// TwinCAT 3 PLC project Untitled1
// ProgramVersion: 3.1.4023.0
// libraries:
//   Tc2_Standard, * (Beckhoff Automation GmbH)
//   Tc2_System, * (Beckhoff Automation GmbH)
//   Tc2_Utilities, * (Beckhoff Automation GmbH)
//   Tc3_Module, * (Beckhoff Automation GmbH)
// project tree:
//   DUTs/ E_EventType.TcDUT, ST_Event.TcDUT
//   / PlcTask.TcTTO
//   POUs/ EventLogger.TcPOU, FB_CSVPersistentEventStorage.TcPOU, I_PersistentEventStorage.TcIO, MAIN.TcPOU, UpdateEventTimeStampWithSystemTime.TcPOU
// real-time tasks:
//   TASK PlcTask: cycle T#10ms, priority 20, ADS port 350

CONFIGURATION Untitled1
    RESOURCE PLC ON TwinCAT3
        TASK PlcTask(INTERVAL := T#10ms, PRIORITY := 20);
        PROGRAM MAIN WITH PlcTask : MAIN;
    END_RESOURCE
END_CONFIGURATION

// ---- DUTs/E_EventType.TcDUT
{attribute 'qualified_only'}
{attribute 'strict'}
TYPE E_EventType :
(
	Alarm := 0,
	Message := 1
);
END_TYPE

// ---- DUTs/ST_Event.TcDUT
TYPE ST_Event :
STRUCT
	eEventType : E_EventType;
	eEventSeverity : TcEventSeverity;
	nEventIdentity : UDINT;
	sEventText : STRING (255);
	dtTimestamp : DATE_AND_TIME;
END_STRUCT
END_TYPE

// ---- POUs/I_PersistentEventStorage.TcIO
INTERFACE I_PersistentEventStorage

METHOD StoreEvent
VAR_INPUT
	stEvent : ST_Event;
END_VAR
END_METHOD

END_INTERFACE

// ---- POUs/MAIN.TcPOU
PROGRAM MAIN
VAR
	//stThisIsOurFirstInstanceOfAstructure : ST_Event;	
	bBoolean : BOOL := FALSE;
	
	eEventType1 : E_EventType := E_EventType.Alarm;
	eEventSeverity1 : TcEventSeverity := TcEventSeverity.Error ;
	nEventIdentity1 : UDINT := 42;
	sEventText1 : STRING (255) := 'This is a scary event';
	
	CSVPersitentEventStorage : FB_CSVPersistentEventStorage;
	EventLogger : EventLogger (CSVPersitentEventStorage);
	
END_VAR

(*
IF NOT bBoolean THEN
	UpdateEventTimeStampWithSystemTime(stEvent := stThisIsOurFirstInstanceOfAstructure);
	bBoolean := TRUE;
END_IF 
*)

IF bBoolean THEN
	EventLogger.AddEvent (eEventType1, eEventSeverity1, nEventIdentity1, sEventText1);
	bBoolean := FALSE;	
END_IF

CSVPersitentEventStorage ();

END_PROGRAM

// ---- POUs/FB_CSVPersistentEventStorage.TcPOU
FUNCTION_BLOCK FB_CSVPersistentEventStorage IMPLEMENTS I_PersistentEventStorage
VAR
	fbFileOpen : FB_FileOpen := (sPathName := 'C:\Events.log', nMode := FOPEN_MODEAPPEND OR FOPEN_MODETEXT); 
	fbFilePuts : FB_FilePuts;
	fbFileClose : FB_FileClose;
	eWriteState : (FILE_OPEN_TRIGGER, FILE_OPEN, WAIT_FOR_EVENT, WRITE_EVENT_TRIGGER, WRITE_EVENT, FILE_CLOSE_TRIGGER, FILE_CLOSE, ERROR);
	stEventWrittenToFile : ST_event;
	CsvString : T_MaxString;
END_VAR

CASE eWriteState OF
	
	FILE_OPEN_TRIGGER: 
		fbFileOpen (bExecute := TRUE);
		eWriteState := FILE_OPEN;
	
	FILE_OPEN :
		fbFileOpen(bExecute := FALSE);
		IF fbFileOpen.bError THEN
			eWriteState := ERROR;
		ELSIF NOT fbFileOpen.bBusy AND fbFileOpen.hFile <> 0 THEN
			eWriteState := WAIT_FOR_EVENT;
		END_IF
		
	WAIT_FOR_EVENT:
	
	 	//DO nothing
	WRITE_EVENT_TRIGGER :
		CsvString := CreateCsvString(stEvent := stEventWrittenToFile);
		fbFilePuts (bExecute := TRUE,
					sLine := CsvString,
					hFile := fbFileOpen.hFile);
		eWriteState := WRITE_EVENT;
	
	WRITE_EVENT :
		fbFilePuts(bExecute := FALSE);
		IF fbFilePuts.bError THEN
			eWriteState := ERROR;
		ELSIF NOT fbFilePuts.bBusy THEN
			eWriteState := FILE_CLOSE_TRIGGER;		
		END_IF
		
	FILE_CLOSE_TRIGGER :
		fbFileClose (bExecute := TRUE,
					 hfile := fbFileOpen.hFile);
		eWriteState := FILE_CLOSE;
		
	FILE_CLOSE :
		fbFileClose (bExecute := FALSE);
		IF fbfileClose.bError THEN
			eWriteState := ERROR;
		ELSIF NOT fbfileClose.bBusy THEN
			eWriteState := FILE_OPEN_TRIGGER;
		END_IF
		
	
	ERROR : 
	
	//DO nothing
	
END_CASE

METHOD PRIVATE CreateCsvString : T_MaxString
VAR_INPUT
	stEvent : REFERENCE TO ST_Event;
END_VAR
VAR
	TempString: T_MaxString;
END_VAR
TempString := TO_STRING (stEvent.eEventType);
TempString := CONCAT (STR1 := TempString, STR2 := ',');
TempString := CONCAT (STR1 := TempString, STR2 := TO_STRING(stEvent.eEventSeverity));
TempString := CONCAT (STR1 := TempString, STR2 := ',');
TempString := CONCAT (STR1 := TempString, STR2 := TO_STRING(stEvent.nEventIdentity));
TempString := CONCAT (STR1 := TempString, STR2 := ',');
TempString := CONCAT (STR1 := TempString, STR2 := stEvent.sEventText);	
TempString := CONCAT (STR1 := TempString, STR2 := ',');
TempString := CONCAT (STR1 := TempString, STR2 := TO_STRING(stEvent.dtTimestamp));
TempString := CONCAT (STR1 := TempString, STR2 := '$n');

CreateCsvString := TempString;
END_METHOD

{warning 'add method implementation '}
METHOD StoreEvent
VAR_INPUT
	stEvent	: ST_Event;
END_VAR
IF eWriteState = WAIT_FOR_EVENT THEN
	eWriteState := WRITE_EVENT_TRIGGER;
	stEventWrittenToFile := stEvent;
END_IF
END_METHOD

END_FUNCTION_BLOCK

// ---- POUs/EventLogger.TcPOU
FUNCTION_BLOCK EventLogger

VAR
	EventBuffer : ARRAY [1..MAXIMUM_SIZE_OF_EVENT_BUFFER] OF ST_Event; 
	CurrentEventBufferIndex : INT := 0;
	_PersistentEventStorage : I_PersistentEventStorage;
END_VAR
VAR CONSTANT
	MAXIMUM_SIZE_OF_EVENT_BUFFER : INT := 100; 
END_VAR

(*Returns TRUE if add was succesful and FALSE if buffer is full *)

METHOD PUBLIC AddEvent : BOOL
VAR_INPUT
	eEventType : E_EventType;
	eEventSeverity : TcEventSeverity;
	nEventIdentity : UDINT;
	sEventText : STRING (255);
END_VAR
IF NOT IsEventBufferFull() THEN
	CurrentEventBufferIndex := CurrentEventBufferIndex + 1;
	EventBuffer[CurrentEventBufferIndex].eEventType := eEventType;
	EventBuffer[CurrentEventBufferIndex].eEventSeverity := eEventSeverity;
	EventBuffer[CurrentEventBufferIndex].nEventIdentity := nEventIdentity;
	EventBuffer[CurrentEventBufferIndex].sEventText := sEventText;
	UpdateEventTimeStampWithSystemTime(stEvent := EventBuffer[CurrentEventBufferIndex]);
	AddEvent := TRUE;
ELSE
	AddEvent := FALSE;
END_IF

//Here we want ti stor the event persistentlty
_PersistentEventStorage.StoreEvent(stEvent := EventBuffer[CurrentEventBufferIndex]);
END_METHOD

METHOD FB_init : BOOL
VAR_INPUT
	bInitRetains : BOOL; // if TRUE, the retain variables are initialized (warm start / cold start)
	bInCopyCode : BOOL;  // if TRUE, the instance afterwards gets moved into the copy code (online change)
	iPersistentEventStorage : I_PersistentEventStorage;
END_VAR
_PersistentEventStorage := iPersistentEventStorage;
END_METHOD

METHOD PRIVATE IsEventBufferFull : BOOL
IF (CurrentEventBufferIndex +1) > MAXIMUM_SIZE_OF_EVENT_BUFFER THEN
	IsEventBufferFull := TRUE;
ELSE
	IsEventBufferFull := FALSE;
END_IF
END_METHOD

END_FUNCTION_BLOCK

// ---- POUs/UpdateEventTimeStampWithSystemTime.TcPOU
FUNCTION UpdateEventTimeStampWithSystemTime
VAR_INPUT
	stEvent : REFERENCE TO ST_Event;
END_VAR
VAR
fbGETSYSTEMTIME : GETSYSTEMTIME;


stFileTime : T_FILETIME;

END_VAR

fbGETSYSTEMTIME(timeLoDW => stFileTime.dwLowDateTime , 
				timeHiDW => stFileTime.dwHighDateTime);
				
stEvent.dtTimestamp := FILETIME_TO_DT(fileTime := stFileTime);

END_FUNCTION
